TYPE ServicesTimingSerialInfoStatuses :
STRUCT
	portHealthStatus: HealthStatus;
	transmissionHealthStatus: HealthStatus;
	checksumHealthStatus: HealthStatus;
	healthStatus: HealthStatus;
END_STRUCT
END_TYPE

(* stored: Version 1.1.0.1, ProductVersion 3.1.4019.2
   DUT ServicesTimingSerialInfoStatuses: Id {c39c4bbf-56bf-4fa9-9200-c92021358eaa} *)
